PROGRAM PRG_Camming
VAR_INPUT
END_VAR
VAR_OUTPUT
END_VAR
VAR
	nState: INT;
	bExecute: BOOL;
	bWriteDoneButton: BOOL;
	ResetButton: BOOL;
END_VAR


MotionFunction[1].FunctionType	:=	MOTIONFUNCTYPE_SINUSLINIE;
MotionFunction[2].FunctionType	:=	MOTIONFUNCTYPE_SINUSLINIE;
MotionFunction[3].FunctionType	:=	MOTIONFUNCTYPE_SINUSLINIE;
MotionFunction[4].FunctionType	:=	MOTIONFUNCTYPE_SINUSLINIE;
MotionFunction[5].FunctionType	:=	MOTIONFUNCTYPE_SINUSLINIE;
MotionFunction[6].FunctionType	:=	MOTIONFUNCTYPE_SINUSLINIE;


CAMTABLE.TableType	:= MC_TABLETYPE_MOTIONFUNCTION;
CAMTABLE.pArray		:= ADR(MotionFunction);
CAMTABLE.ArraySize	:= SIZEOF(MotionFunction);
CAMTABLE.NoOfColumns:= 1;
CAMTABLE.NoOfRows	:= SIZEOF(MotionFunction)/SIZEOF(MotionFunction[1]);


AxisInterface1.IN.bPower	:=	TRUE;
AxisInterface1.IN.nOverride	:=	100;

AxisInterface2.IN.bPower	:=	TRUE;
AxisInterface2.IN.nOverride	:=	100;



CASE nState	OF
	
	0:
		IF bExecute	
		AND AxisInterface1.OUT.bPowerEnabled 
		AND AxisInterface2.OUT.bPowerEnabled	THEN
			Axisinterface1.IN.bStop		:=	FALSE;
			Axisinterface2.IN.bStop		:=	FALSE;
			
			IF NOT AxisInterface1.OUT.bStopActive AND NOT AxisInterface2.OUT.bStopActive THEN
							nState:=5;
			END_IF
			
		END_IF
		
		
	5:
		AxisInterface1.IN.bCamIN	:=TRUE;
		AxisInterface1.IN.nCamTableID	:=	1;
		
		IF AxisInterface1.OUT.bCamINDone	THEN			
			AxisInterface1.IN.bCamIN	:=FALSE;
			nState						:=	10;			
		END_IF
	
	10:
			

			IF AxisInterface1.OUT.bPowerEnabled 
			AND AxisInterface2.OUT.bPowerEnabled	THEN
			
	
			
			AxisInterface1.IN.fPos		:=	18000;
			AxisInterface1.IN.fVelocity	:=	1500;
		
			AxisInterface1.IN.bAbs		:=	TRUE;			
			nstate	:=	20;
			
			
		
		ELSIF Axisinterface1.OUT.bAbsErr	THEN
			nState	:=	999;
		END_IF
		
	
			
			20:	
		IF AxisInterface1.OUT.bAbsBusy
		AND NOT AxisInterface1.OUT.bAbsErr	THEN
			
			nState	:=	30;
			
			ELSIF Axisinterface1.OUT.bAbsErr	THEN
				nState	:=	999;
			END_IF
			
	
	30:
		IF AxisInterface1.OUT.bAbsDone
		AND NOT AxisInterface1.OUT.bAbsErr	THEN
		
		AxisInterface1.IN.bAbs		:=	FALSE;
		AxisInterface1.IN.bCamOUT	:=	TRUE;
		AxisInterface1.IN.bCamIN	:=FALSE;

		nState	:=	31;
		
			
		ELSIF Axisinterface1.OUT.bAbsErr	THEN
	//	nState	:=	999;
			
		END_IF
		
		31:
			IF AxisInterface1.OUT.bCamOUTDone	THEN
				nState	:=	32;
				AxisInterface1.IN.bCamOUT	:=	FALSE;
			END_IF
		
	32:
		AxisInterface1.IN.bRead	:=	TRUE;
		AxisInterface1.IN.nCamTableIdWr	:=	1;

			IF AxisInterface1.OUT.bReadDone THEN
				nState	:=40;
				AxisInterface1.IN.bRead	:= FALSE;		
			END_IF
		
		
	40:
	
		MotionFunction[1].SlavePos	:= arrSlavePos[1];
		MotionFunction[2].SlavePos	:= arrSlavePos[2];
		MotionFunction[3].SlavePos	:= arrSlavePos[3];
		MotionFunction[4].SlavePos	:= arrSlavePos[4];
		MotionFunction[5].SlavePos	:= arrSlavePos[5];
		MotionFunction[6].SlavePos	:= arrSlavePos[6];
		MotionFunction[7].SlavePos	:= arrSlavePos[7];
		
		MotionFunction[1].MasterPos	:= 0;
		MotionFunction[2].MasterPos	:= 60;
		MotionFunction[3].MasterPos	:= 120;
		MotionFunction[4].MasterPos	:= 180;
		MotionFunction[5].MasterPos	:= 240;
		MotionFunction[6].MasterPos	:= 300;
		MotionFunction[7].MasterPos	:= 360;
		
	
		
		
		
AxisInterface1.IN.bWrite	:=	bWriteDoneButton;
		
		IF AxisInterface1.OUT.bWriteDone	 THEN
			AxisInterface1.IN.bWrite	:= FALSE;
			nState					:= 50;		
		END_IF
	
	50:
		
		IF AxisInterface1.OUT.bPowerEnabled 
		AND AxisInterface1.OUT.bPowerEnabled
		AND NOT AxisInterface1.OUT.bAbsErr	THEN
		
			AxisInterface1.IN.fPos		:=	0;
			AxisInterface1.IN.fVelocity	:=	2000;
			AxisInterface1.IN.bAbs		:=	TRUE;
			
			nState						:=	60;
			
	
		ELSIF Axisinterface1.OUT.bAbsErr	THEN
			nState	:=	999;
		END_IF
	
	60:
	
		IF AxisInterface1.OUT.bAbsBusy
		AND NOT AxisInterface1.OUT.bAbsErr	THEN
			
			nState	:=	70;
			AxisInterface1.IN.bAbs		:=	FALSE;
			
		ELSIF Axisinterface1.OUT.bAbsErr	THEN
			nState	:=	999;
		END_IF
			

	70:
		
		IF AxisInterface1.OUT.babsdone
		AND NOT AxisInterface1.OUT.bAbsErr	THEN
		
			nState	:=	0;

			
		ELSIF Axisinterface1.OUT.bAbsErr	THEN
				nState	:=	999;
		END_IF
		
END_CASE

IF NOT bExecute THEN
	
	AxisInterface1.IN.bStop	:=	TRUE;
	AxisInterface2.IN.bStop	:=	TRUE;

	AxisInterface1.IN.bAbs	:=	FALSE;

		
END_IF
	
	
IF ResetButton THEN


	AxisInterface1.IN.bReset	:=	TRUE;	
	
	IF AxisInterface1.OUT.bResetDone	THEN
		nState	:=	0;
		bExecute	:=	FALSE;
	END_IF

END_IF

END_PROGRAM

(* stored: Version 1.1.0.1, ProductVersion 3.1.4022.18
   POU PRG_Camming: Id {9300bb5a-f69c-4e7e-a1f0-9eaf896a99ee}, SpecialFunc None *)
